TYPE E_EcCommState :
(
	eEcState_UNDEFINED := 0,
	eEcState_INIT := 1,
	eEcState_PREOP := 2,
	eEcState_BOOT := 3,
	eEcState_SAFEOP := 4,
	eEcState_OP := 8
);
END_TYPE

(* stored: Version 1.1.0.1, ProductVersion 3.1.0.12
   DUT E_EcCommState: Id {b34abcf1-8693-4cad-ab2a-3160af290cdb} *)
